(* IEC 61131-3 sources: kst/tests, 86 files *)

(* ---- f.1.st ---- *)
FUNCTION WEIGH : INT
  VAR_INPUT
    weigh_command : BOOL;
    gross_weight : INT ;
    tare_weight : INT ;
  END_VAR

IF weigh_command THEN
  WEIGH := gross_weight - tare_weight;
END_IF ;
END_FUNCTION

(* ---- f.11.st ---- *)
FUNCTION ALRMINT : BOOL
VAR_INPUT
  IN:INT;
  THI:INT ;
  TLO:INT  ;
END_VAR
VAR_OUTPUT
  HI: BOOL;
  LO: BOOL;
END_VAR
HI := IN > THI ;

LO := IN < THL ;
ALRMINT := THI OR THL ;
END_FUNCTION

(* ---- f10.st ---- *)
FUNCTION SIMPLE_FUN : REAL
    VAR_INPUT
  		A, B : REAL ;
      	C : REAL := 1.0;
  	END_VAR
  	VAR_IN_OUT COUNT : INT ; END_VAR
  	VAR COUNTP1 : INT ; END_VAR

  	COUNTP1 := ADD(COUNT,1);
  	COUNT := COUNTP1 ;
    SIMPLE_FUN := A*B/C;
END_FUNCTION

(* ---- f22.st ---- *)
FUNCTION Test : BOOL
	VAR_INPUT
		SUM : INT;
		FLAG : BOOL;
	END_VAR
	VAR
		I, J : INT;
	END_VAR

	SUM := 0 ;
	FOR I := 1 TO 3 DO
		FOR J := 1 TO 2 DO
			IF FLAG THEN EXIT ; END_IF
			SUM := SUM + J ;
		END_FOR ;
		SUM := SUM + I ;
	END_FOR ;
END_FUNCTION

(* ---- f5.st ---- *)
FUNCTION Test : INT
	VAR_INPUT
		B, C, D : INT;
		X : INT;
	END_VAR
	VAR_OUTPUT
		A : INT;
		NO_ERR : BOOL;
	END_VAR

	A := ADD(B, C, D);
	A := SHL(IN:=B, N:=C);
	A := SHL(EN:=ENABLE, IN:=B, N:=C, NOT ENO=>NO_ERR);
	A := INC(V:=X);

END_FUNCTION

(* ---- t19-1.st ---- *)
FUNCTION Test : INT
	VAR_INPUT
		B, COND, TEMPL : INT;
	END_VAR
	VAR_OUTPUT
		A : INT;
	END_VAR

	A := LIMIT(EN:=COND, IN:=B, MX:=5, ENO=>TEMPL);

END_FUNCTION

(* ---- t19-2.st ---- *)
FUNCTION Test : INT
	VAR_INPUT
		B : INT;
	END_VAR
	VAR_OUTPUT
		A : INT;
	END_VAR

	A := LIMIT(1, B, 5);

END_FUNCTION

(* ---- t20-3a.st ---- *)
FUNCTION SIMPLE_FUN : REAL
    VAR_INPUT
  		A, B : REAL ;
      	C : REAL := 1.0;
  	END_VAR
  	VAR_IN_OUT COUNT : INT ; END_VAR
  	VAR COUNTP1 : INT ; END_VAR

  	COUNTP1 := ADD(COUNT,1);
  	COUNT := COUNTP1 ;
    SIMPLE_FUN := A*B/C;
END_FUNCTION

(* ---- t56-1.st ---- *)
FUNCTION Test : INT
	VAR_INPUT
		B : INT;
	END_VAR
	VAR_OUTPUT
		A, CV : INT;
		C : REAL;
	END_OUTPUT

	A := B;
	CV := CV+1;
	C := SIN(X);

END_FUNCTION

(* ---- t56-4.st ---- *)
FUNCTION Test : BOOL
	VAR_INPUT
		A, B, C : REAL;
	END_VAR
	VAR_OUTPUT
		D, X1, X2 : REAL;
		NROOTS : INT;
	END_VAR

	D := B*B - 4*A*C ;
	IF D < 0.0 THEN NROOTS := 0 ;
	ELSIF D = 0.0 THEN
		NROOTS := 1 ;
		X1 := - B/(2.0*A) ;
	ELSE
		NROOTS := 2 ;
		X1 := (- B + SQRT(D))/(2.0*A) ;
		X2 := (- B - SQRT(D))/(2.0*A) ;
	END_IF ;
END_FUNCTION

(* ---- t56-6.st ---- *)
FUNCTION Test : BOOL
	VAR_INPUT
		I, J : INT;
	END_VAR

	J := 101 ;
	FOR I := 1 TO 100 BY 2 DO
		IF I MOD 2 == 0 THEN
			J := I ;
			EXIT ;
		END_IF ;
	END_FOR ;
END_FUNCTION

(* ---- t56-7.st ---- *)
FUNCTION Test : BOOL
	VAR_INPUT
		J : INT;
	END_VAR

	J := 1;
	WHILE J <= 100 DO
		J := J+2 ;
	END_WHILE ;
END_FUNCTION

(* ---- t56-8.st ---- *)
FUNCTION Test : BOOL
	VAR_INPUT
		J : INT;
	END_VAR

	J := -1 ;
	REPEAT
	  J := J+2 ;
	UNTIL J = 101
	END_REPEAT ;
END_FUNCTION

(* ---- f.2.st ---- *)
FUNCTION_BLOCK CMD_MONITOR
 VAR_INPUT AUTO_CMD : BOOL ;
          AUTO_MODE : BOOL ;
            MAN_CMD : BOOL ;
        MAN_CMD_CHK : BOOL ;
          T_CMD_MAX : REAL ;
               FDBK : BOOL ;
                ACK : BOOL ;
 END_VAR
 VAR_OUTPUT CMD : BOOL ;
           ALRM : BOOL ;
 END_VAR
 VAR CMD_TMR : TON ;
     ALRM_FF : SR ;
 END_VAR

 CMD := AUTO_CMD & AUTO_MODE
          OR MAN_CMD & NOT MAN_CMD_CHK & NOT AUTO_MODE ;
    CMD_TMR (IN := CMD, PT := T_CMD_MAX);
    ALRM_FF (S1 := CMD_TMR.Q & NOT FDBK, R := ACK);
    ALRM := ALRM_FF.Q1;

END_FUNCTION_BLOCK

(* ---- f.3.st ---- *)
FUNCTION_BLOCK FWD_REV_MON
VAR_INPUT AUTO : BOOL ;
  ACK : BOOL ;
  AUTO_FWD : BOOL ;
  MAN_FWD : BOOL ;
  MAN_FWD_CHK : BOOL ;
  T_FWD_MAX : TIME ;
  FWD_FDBK : BOOL ;

  AUTO_REV : BOOL ;
  MAN_REV : BOOL ;
  MAN_REV_CHK : BOOL ;
  T_REV_MAX : TIME ;
  REV_FDBK : BOOL ;
END_VAR
VAR_OUTPUT KLAXON : BOOL ;
  FWD_REV_ALRM : BOOL;
  FWD_CMD : BOOL ;
  FWD_ALRM : BOOL ;
  REV_CMD : BOOL ;
  REV_ALRM : BOOL ;
END_VAR
VAR FWD_MON : CMD_MONITOR;
  REV_MON : CMD_MONITOR;
  FWD_REV_FF : SR ;
END_VAR

  FWD_MON    (AUTO_MODE   := AUTO,
              ACK         := ACK,
              AUTO_CMD    := AUTO_FWD,
              MAN_CMD     := MAN_FWD,
              MAN_CMD_CHK := MAN_FWD_CHK,
              T_CMD_MAX   := T_FWD_MAX,
              FDBK        := FWD_FDBK);
  REV_MON    (AUTO_MODE   := AUTO,
              ACK         := ACK,
              AUTO_CMD    := AUTO_REV,
              MAN_CMD     := MAN_REV,
              MAN_CMD_CHK := MAN_REV_CHK,
              T_CMD_MAX   := T_REV_MAX,
              FDBK        := REV_FDBK);
  FWD_REV_FF (S1 := FWD_MON.CMD & REV_MON.CMD, R := ACK);

  FWD_REV_ALRM := FWD_REV_FF.Q1;
  FWD_CMD := FWD_MON.CMD & NOT FWD_REV_ALRM;
  FWD_ALRM := FWD_MON.ALRM;
  REV_CMD := REV_MON.CMD & NOT FWD_REV_ALRM;
  REV_ALRM := REV_MON.ALRM;
  KLAXON := FWD_ALRM OR REV_ALRM OR FWD_REV_ALRM;
END_FUNCTION_BLOCK

(* ---- f.4.st ---- *)
FUNCTION_BLOCK STACK_INT
  VAR_INPUT PUSH, POP: BOOL;
            R1 : BOOL ;
            IN : INT ;
            N  : INT ;
  END_VAR
  VAR_OUTPUT EMPTY : BOOL := 1 ;
             OFLO  : BOOL := 0 ;
             OUT   : INT  := 0 ;
  END_VAR
  VAR STK : ARRAY[0..127] OF INT;
      NI : INT :=128  ;
      PTR : INT := -1 ;
  END_VAR

    IF R1 THEN
       OFLO := 0; EMPTY := 1; PTR := -1;
       NI := LIMIT (MN:=1,IN:=N,MX:=128); OUT := 0;
    ELSIF POP & NOT EMPTY THEN
       OFLO := 0; PTR := PTR-1; EMPTY := PTR < 0;
       IF EMPTY THEN OUT := 0;
       ELSE OUT := STK[PTR];
       END_IF ;
    ELSIF PUSH & NOT OFLO THEN
       EMPTY := 0; PTR := PTR+1; OFLO := (PTR = NI);
       IF NOT OFLO THEN OUT := IN ; STK[PTR] := IN;
       ELSE OUT := 0;
       END_IF ;
    END_IF ;
END_FUNCTION_BLOCK

(* ---- f.6.1.st ---- *)
FUNCTION_BLOCK LAG1
   VAR_INPUT
     RUN : BOOL ;
     XIN : REAL ;
     TAU : REAL ;
     CYCLE : REAL ;
   END_VAR
   VAR_OUTPUT XOUT : REAL ; END_VAR
   VAR K : REAL ;
   END_VAR
   IF RUN THEN XOUT := XOUT + K * (XIN - XOUT) ;
   ELSE XOUT := XIN ;
        K := CYCLE /(CYCLE + TAU) ;
   END_IF ;
END_FUNCTION_BLOCK

(* ---- f.6.10.st ---- *)
FUNCTION_BLOCK PID
   VAR_INPUT
     AUTO : BOOL ;
     PV : REAL ;
     SP : REAL ;
     X0 : REAL ;

     KP : REAL ;
     TR : REAL ;
     TD : REAL ;
     CYCLE : REAL ;
   END_VAR
   VAR_OUTPUT XOUT : REAL; END_VAR
   VAR ERROR : REAL ;
       ITERM : INTEGRAL ;
       DTERM : DERIVATIVE ;
   END_VAR
   ERROR := PV - SP ;

   ITERM (RUN := AUTO, R1 := NOT AUTO, XIN := ERROR,
          X0 := TR * (X0 - ERROR), CYCLE := CYCLE) ;
   DTERM (RUN := AUTO, XIN := ERROR, CYCLE := CYCLE) ;
   XOUT := KP * (ERROR + ITERM.XOUT/TR + DTERM.XOUT*TD) ;
 END_FUNCTION_BLOCK

(* ---- f.6.11.st ---- *)
FUNCTION_BLOCK DIFFEQ
   VAR_INPUT
     RUN : BOOL ;
     XIN : REAL ;
     A : ARRAY[1..127] OF REAL ;
     M : INT ;
     B : ARRAY[0..127] OF REAL ;
     N : INT ;
   END_VAR
   VAR_OUTPUT XOUT : REAL := 0.0 ; END_VAR
   VAR
     XI : ARRAY [0..127] OF REAL ;
     XO : ARRAY [0..127] OF REAL ;
     I : INT ;
   END_VAR
   XO[0] := XOUT ; XI[0] := XIN ;
   XOUT := B[0] * XIN ;
   IF RUN THEN
      FOR I := M TO 1 BY -1 DO
          XOUT := XOUT + A[I] * XO[I] ; XO[I] := XO[I-1];
      END_FOR;
      FOR I := N TO 1 BY -1 DO
          XOUT := XOUT + B[I] * XI[I] ; XI[I] := XI[I-1];
      END_FOR;
   ELSE
      FOR I := 1 TO M DO XO[I] := 0.0; END_FOR;
      FOR I := 1 TO N DO XI[I] := 0.0; END_FOR;
   END_IF ;
 END_FUNCTION_BLOCK

(* ---- f.6.12.st ---- *)
 FUNCTION_BLOCK RAMP
   VAR_INPUT
     RUN : BOOL ;
     X0,X1 : REAL ;
     TR : REAL ;
     CYCLE : REAL ;
   END_VAR
   VAR_OUTPUT
     BUSY : BOOL ;
     XOUT : REAL := 0.0 ;
   END_VAR
   VAR XI : REAL ;
       T : REAL := 0.0;
   END_VAR
   BUSY := RUN ;
   IF RUN THEN
      IF T >= TR THEN BUSY := 0 ; XOUT := X1 ;
      ELSE XOUT := XI + (X1-XI) * T
                                / TR ;
           T := T + CYCLE ;
      END_IF ;
   ELSE XOUT := X0 ; XI := X0 ; T := 0.0 ;
   END_IF ;
 END_FUNCTION_BLOCK

(* ---- f.6.13.st ---- *)
FUNCTION_BLOCK TRANSFER
 VAR_INPUT
   AUTO : BOOL ;
   XIN : REAL ;
   FASTRATE, SLOWRATE : REAL ;
   FASTUP, SLOWUP,
   FASTDOWN, SLOWDOWN : BOOL;
   CYCLE : TIME ;
 END_VAR
 VAR_OUTPUT XOUT : REAL ; END_VAR
 VAR XFERRAMP : INTEGRAL ;
     RAMPRATE : REAL ;
 END_VAR
 RAMPRATE := 0.0 ;
 IF NOT AUTO THEN
  IF FASTUP THEN RAMPRATE := FASTRATE; END_IF;
  IF SLOWUP THEN RAMPRATE := RAMPRATE + SLOWRATE; END_IF;
  IF FASTDOWN THEN RAMPRATE := RAMPRATE - FASTRATE; END_IF;
  IF SLOWDOWN THEN RAMPRATE := RAMPRATE - SLOWRATE; END_IF;
 END_IF ;
 XFERRAMP (RUN := 1, CYCLE := CYCLE, R1 := AUTO,
            XIN := RAMPRATE, X0 := XIN) ;
 XOUT := XFERRAMP.XOUT;
END_FUNCTION_BLOCK

(* ---- f.6.2.st ---- *)
FUNCTION_BLOCK DELAY
  VAR_INPUT
    RUN : BOOL ;
    XIN : REAL ;
    N   : INT ;
  END_VAR
  VAR_OUTPUT XOUT : REAL; END_VAR
  VAR X : ARRAY [0..127]
               OF REAL;
      I, IXIN, IXOUT : INT := 0;
  END_VAR
  IF RUN THEN IXIN := MOD(IXIN + 1, 128) ; X[IXIN] := XIN ;
              IXOUT := MOD(IXOUT + 1, 128) ; XOUT := X[IXOUT];
  ELSE XOUT := XIN ; IXIN := N ; IXOUT := 0;
       FOR I := 0 TO N DO X[I] := XIN; END_FOR;
  END_IF ;
END_FUNCTION_BLOCK

(* ---- f.6.3.st ---- *)
FUNCTION_BLOCK AVERAGE
   VAR_INPUT
     RUN : BOOL ;
     XIN : REAL ;
     N   : INT ;
   END_VAR
   VAR_OUTPUT XOUT : REAL ; END_VAR
   VAR SUM  : REAL := 0.0;
       FIFO : DELAY ;
   END_VAR
   SUM := SUM - FIFO.XOUT ;
   FIFO (RUN := RUN , XIN := XIN, N := N) ;
   SUM := SUM + FIFO.XOUT ;
   IF RUN THEN XOUT := SUM/N ;
   ELSE SUM := N*XIN ; XOUT := XIN ;
   END_IF ;
 END_FUNCTION_BLOCK

(* ---- f.6.4.st ---- *)
FUNCTION_BLOCK INTEGRAL
   VAR_INPUT
     RUN : BOOL ;
     R1 : BOOL ;
     XIN : REAL ;
     X0  : REAL ;
     CYCLE : REAL ;
   END_VAR
   VAR_OUTPUT
     Q : BOOL ;
     XOUT : REAL ;
   END_VAR
   Q := NOT R1 ;
   IF R1 THEN XOUT := X0 ;
   ELSIF RUN THEN XOUT := XOUT + XIN * TIME_TO_REAL(CYCLE);
   END_IF ;
 END_FUNCTION_BLOCK

(* ---- f.6.5.st ---- *)
FUNCTION_BLOCK DERIVATIVE
   VAR_INPUT
     RUN : BOOL ;
     XIN : REAL ;
     CYCLE : REAL ;
   END_VAR
   VAR_OUTPUT
     XOUT : REAL ;
   END_VAR
   VAR X1, X2, X3 : REAL ; END_VAR
   IF RUN THEN
      XOUT := (3.0 * (XIN - X3) + X1 - X2)
              / (10.0 * CYCLE) ;
      X3 := X2 ; X2 := X1 ; X1 := XIN ;
   ELSE XOUT := 0.0; X1 := XIN ; X2 := XIN ; X3 := XIN ;
   END_IF ;
 END_FUNCTION_BLOCK

(* ---- f.6.6.st ---- *)
 FUNCTION_BLOCK HYSTERESIS
  VAR_INPUT XIN1, XIN2, EPS : REAL; END_VAR
  VAR_OUTPUT Q : BOOL := 0; END_VAR
  IF Q THEN IF XIN1 < (XIN2 - EPS) THEN Q := 0; END_IF ;
  ELSIF XIN1 > (XIN2 + EPS) THEN Q := 1 ;
  END_IF ;
END_FUNCTION_BLOCK

(* ---- f19.st ---- *)
FUNCTION_BLOCK A
	VAR_OUTPUT
		y1 : UINT ; y2 : BYTE ;
	END_VAR
END_FUNCTION_BLOCK

FUNCTION_BLOCK B
	VAR_INPUT
		b1 : UINT ; b2 : BYTE ;
	END_VAR
END_FUNCTION_BLOCK

FUNCTION_BLOCK C
	VAR_OUTPUT c1 : BOOL ; END_VAR
	VAR C2 AT %Q*: BYTE;
		C3: INT;
	END_VAR
END_FUNCTION_BLOCK

FUNCTION_BLOCK D
	VAR_INPUT d1 : BOOL ; END_VAR
	VAR_OUTPUT y2 : INT ; END_VAR
END_FUNCTION_BLOCK

PROGRAM F
	VAR_INPUT  x1 : BOOL ;  x2 : UINT ; END_VAR
	VAR_OUTPUT y1 : BYTE ; END_VAR
	VAR COUNT: INT; TIME1: TON; END_VAR
END_PROGRAM

PROGRAM G
	VAR_OUTPUT out1 : UINT ;  END_VAR
	VAR_EXTERNAL z1 : BYTE ;  END_VAR
	VAR  FB1 : A ;  FB2 : B ; END_VAR
	FB1();
	out1 := FB1.y1;
	z1 := FB1.y2;
    FB2(b1 := FB1.y1, b2 := FB1.y2) ;
END_PROGRAM

PROGRAM H
	VAR_OUTPUT HOUT1: INT ;  END_VAR
	VAR  FB1 : C ;  FB2 : D ; END_VAR
	FB1();
	FB2(d1:=TRUE);
	HOUT1 := FB2.y2;
END_PROGRAM

(* ---- hc-t-171.st ---- *)
PROGRAM temp
  VAR
    I1,I2,I3,I4:INT;
    B1,B2,B3,B4,B5,B6,B7:BOOL;
    R1,R2,R3,R4:REAL;
  END_VAR

  CMD_MONITOR(AUTO_CMD:=B1,AUTO_MODE:=B2,MAN_CMD:=B3,MAN_CMD_CHK:=B4,FDBK:=B5,ACK:=B6,T_CMD_MAX:=R1);

END_PROGRAM

FUNCTION_BLOCK CMD_MONITOR
 VAR_INPUT AUTO_CMD : BOOL ;
          AUTO_MODE : BOOL ;
            MAN_CMD : BOOL ;
        MAN_CMD_CHK : BOOL ;
          T_CMD_MAX : REAL ;
               FDBK : BOOL ;
                ACK : BOOL ;
 END_VAR
 VAR_OUTPUT CMD : BOOL ;
           ALRM : BOOL ;
 END_VAR
 VAR CMD_TMR : TON ;
     ALRM_FF : SR ;
 END_VAR

 CMD := AUTO_CMD & AUTO_MODE
          OR MAN_CMD & NOT MAN_CMD_CHK & NOT AUTO_MODE ;
    CMD_TMR (IN := CMD, PT := T_CMD_MAX);
    ALRM_FF (S1 := CMD_TMR.Q & NOT FDBK, R := ACK);
    ALRM := ALRM_FF.Q1;

END_FUNCTION_BLOCK

(* ---- hc-t-178.st ---- *)
PROGRAM temp
  VAR
    I1,I2,I3,I4:INT;
    B1,B2,B3:BOOL;
    R0,R2,R3,R4:REAL;
  END_VAR

  STACK_INT(PUSH:=B1,POP:=B2,R1:=B3,IN:=I1,N:=I2);

END_PROGRAM

FUNCTION_BLOCK STACK_INT
  VAR_INPUT PUSH, POP: BOOL R_EDGE;
            R1 : BOOL ;
            IN : INT ;
            N  : INT ;
  END_VAR
  VAR_OUTPUT EMPTY : BOOL := 1 ;
             OFLO  : BOOL := 0 ;
             OUT   : INT  := 0 ;
  END_VAR
  VAR STK : ARRAY[0..127] OF INT;
      NI : INT :=128  ;
      PTR : INT := -1 ;
  END_VAR

    IF R1 THEN
       OFLO := 0; EMPTY := 1; PTR := -1;
       NI := LIMIT (MN:=1,IN:=N,MX:=128); OUT := 0;
    ELSIF POP & NOT EMPTY THEN
       OFLO := 0; PTR := PTR-1; EMPTY := PTR < 0;
       IF EMPTY THEN OUT := 0;
       ELSE OUT := STK[PTR];
       END_IF ;
    ELSIF PUSH & NOT OFLO THEN
       EMPTY := 0; PTR := PTR+1; OFLO := (PTR = NI);
       IF NOT OFLO THEN OUT := IN ; STK[PTR] := IN;
       ELSE OUT := 0;
       END_IF ;
    END_IF ;
END_FUNCTION_BLOCK

(* ---- hc-t-187.st ---- *)
PROGRAM temp
  VAR
    I1,I2,I3,I4:INT;
    B1,B2,B3:BOOL;
    R1,R2,R3,R4:REAL;
  END_VAR

  LAG1(RUN:=B1,XIN:=R1,TAU:=R2,CYCLE:=R3)
  DELAY(RUN:=B1,XIN:=R1,TAU:=R2,CYCLE:=R3)

END_PROGRAM

FUNCTION_BLOCK LAG1
   VAR_INPUT
     RUN : BOOL ;
     XIN : REAL ;
     TAU : REAL ;
     CYCLE : REAL ;
   END_VAR
   VAR_OUTPUT XOUT : REAL ; END_VAR
   VAR K : REAL ;
   END_VAR
   IF RUN THEN XOUT := XOUT + K * (XIN - XOUT) ;
   ELSE XOUT := XIN ;
        K := CYCLE /(CYCLE + TAU) ;
   END_IF ;
 END_FUNCTION_BLOCK

 FUNCTION_BLOCK DELAY
  VAR_INPUT
    RUN : BOOL ;
    XIN : REAL ;
    N   : INT ;
  END_VAR
  VAR_OUTPUT XOUT : REAL; END_VAR
  VAR X : ARRAY [0..127]
               OF REAL;
      I, IXIN, IXOUT : INT := 0;
  END_VAR
  IF RUN THEN IXIN := MOD(IXIN + 1, 128) ; X[IXIN] := XIN ;
              IXOUT := MOD(IXOUT + 1, 128) ; XOUT := X[IXOUT];
  ELSE XOUT := XIN ; IXIN := N ; IXOUT := 0;
       FOR I := 0 TO N DO X[I] := XIN; END_FOR;
  END_IF ;
END_FUNCTION_BLOCK

(* ---- hc-t-188.st ---- *)
PROGRAM temp
  VAR
    I1,I2,I3,I4:INT;
    B1,B2,B3:BOOL;
    R0,R2,R3,R4:REAL;
  END_VAR

  AVERAGE(RUN:=B1,XIN:=R0,N:=I1);
  INTEGRAL(RUN:=B1,R1:=B2,XIN:=R0,X0:=R2,CYCLE:=R43);

END_PROGRAM

FUNCTION_BLOCK AVERAGE
   VAR_INPUT
     RUN : BOOL ;
     XIN : REAL ;
     N   : INT ;
   END_VAR
   VAR_OUTPUT XOUT : REAL ; END_VAR
   VAR SUM  : REAL := 0.0;
       FIFO : DELAY ;
   END_VAR
   SUM := SUM - FIFO.XOUT ;
   FIFO (RUN := RUN , XIN := XIN, N := N) ;
   SUM := SUM + FIFO.XOUT ;
   IF RUN THEN XOUT := SUM/N ;
   ELSE SUM := N*XIN ; XOUT := XIN ;
   END_IF ;
 END_FUNCTION_BLOCK

FUNCTION_BLOCK INTEGRAL
   VAR_INPUT
     RUN : BOOL ;
     R1 : BOOL ;
     XIN : REAL ;
     X0  : REAL ;
     CYCLE : REAL ;
   END_VAR
   VAR_OUTPUT
     Q : BOOL ;
     XOUT : REAL ;
   END_VAR
   Q := NOT R1 ;
   IF R1 THEN XOUT := X0 ;
   ELSIF RUN THEN XOUT := XOUT + XIN * TIME_TO_REAL(CYCLE);
   END_IF ;
 END_FUNCTION_BLOCK

(* ---- hc-t-189.st ---- *)
PROGRAM temp
  VAR
    I1,I2,I3,I4:INT;
    B1,B2,B3:BOOL;
    R1,R2,R3,R4:REAL;
  END_VAR
  DERIVATIVE(RUN:=B1,XIN:=R1,CYCLE:=R2);
  HYSTERESIS(XIN1:=R3,XIN2:=R4,EPS:=R5);
END_PROGRAM

FUNCTION_BLOCK DERIVATIVE
   VAR_INPUT
     RUN : BOOL ;
     XIN : REAL ;
     CYCLE : REAL ;
   END_VAR
   VAR_OUTPUT
     XOUT : REAL ;
   END_VAR
   VAR X1, X2, X3 : REAL ; END_VAR
   IF RUN THEN
      XOUT := (3.0 * (XIN - X3) + X1 - X2)
              / (10.0 * CYCLE) ;
      X3 := X2 ; X2 := X1 ; X1 := XIN ;
   ELSE XOUT := 0.0; X1 := XIN ; X2 := XIN ; X3 := XIN ;
   END_IF ;
 END_FUNCTION_BLOCK

 FUNCTION_BLOCK HYSTERESIS
  VAR_INPUT XIN1, XIN2, EPS : REAL; END_VAR
  VAR_OUTPUT Q : BOOL := 0; END_VAR
  IF Q THEN IF XIN1 < (XIN2 - EPS) THEN Q := 0; END_IF ;
  ELSIF XIN1 > (XIN2 + EPS) THEN Q := 1 ;
  END_IF ;
END_FUNCTION_BLOCK

(* ---- hc-t-192.st ---- *)
PROGRAM temp
  VAR
    I1,I2,I3,I4:INT;
    B1,B2,B3:BOOL;
    R1,R2,R3,R4,R5,R6,R7:REAL;
  END_VAR

  PID(AUTO:=B1,PV:=R1,SP:=R2,X0:=R3,KP:=R4,TR:=R5,TD:=R6,CYCLE:=R7);

END_PROGRAM

FUNCTION_BLOCK PID
   VAR_INPUT
     AUTO : BOOL ;
     PV : REAL ;
     SP : REAL ;
     X0 : REAL ;

     KP : REAL ;
     TR : REAL ;
     TD : REAL ;
     CYCLE : REAL ;
   END_VAR
   VAR_OUTPUT XOUT : REAL; END_VAR
   VAR ERROR : REAL ;
       ITERM : INTEGRAL ;
       DTERM : DERIVATIVE ;
   END_VAR
   ERROR := PV - SP ;

   ITERM (RUN := AUTO, R1 := NOT AUTO, XIN := ERROR,
          X0 := TR * (X0 - ERROR), CYCLE := CYCLE) ;
   DTERM (RUN := AUTO, XIN := ERROR, CYCLE := CYCLE) ;
   XOUT := KP * (ERROR + ITERM.XOUT/TR + DTERM.XOUT*TD) ;
 END_FUNCTION_BLOCK

(* ---- hc-t-193.st ---- *)
PROGRAM temp
  VAR
    P1,P2:INT;
    P3:REAL;
    P4:BOOL;
  END_VAR

  DIFFEQ(RUN:=P4,XIN:=P3);

END_PROGRAM

FUNCTION_BLOCK DIFFEQ
   VAR_INPUT
     RUN : BOOL ;
     XIN : REAL ;
     A : ARRAY[1..127] OF REAL ;
     M : INT ;
     B : ARRAY[0..127] OF REAL ;
     N : INT ;
   END_VAR
   VAR_OUTPUT XOUT : REAL := 0.0 ; END_VAR
   VAR
     XI : ARRAY [0..127] OF REAL ;
     XO : ARRAY [0..127] OF REAL ;
     I : INT ;
   END_VAR
   XO[0] := XOUT ; XI[0] := XIN ;
   XOUT := B[0] * XIN ;
   IF RUN THEN
      FOR I := M TO 1 BY -1 DO
          XOUT := XOUT + A[I] * XO[I] ; XO[I] := XO[I-1];
      END_FOR;
      FOR I := N TO 1 BY -1 DO
          XOUT := XOUT + B[I] * XI[I] ; XI[I] := XI[I-1];
      END_FOR;
   ELSE
      FOR I := 1 TO M DO XO[I] := 0.0; END_FOR;
      FOR I := 1 TO N DO XI[I] := 0.0; END_FOR;
   END_IF ;
 END_FUNCTION_BLOCK

(* ---- hc-t-194.st ---- *)
PROGRAM temp
  VAR
    I1,I2,I3,I4:INT;
    B1,B2,B3:BOOL;
    R1,R2,R3,R4:REAL;
  END_VAR
  RAMP(RUN:=B1,X0:=R1,X1:=R2,TR:=R3,CYCLE:=R4);

END_PROGRAM

 FUNCTION_BLOCK RAMP
   VAR_INPUT
     RUN : BOOL ;
     X0,X1 : REAL ;
     TR : REAL ;
     CYCLE : REAL ;
   END_VAR
   VAR_OUTPUT
     BUSY : BOOL ;
     XOUT : REAL := 0.0 ;
   END_VAR
   VAR XI : REAL ;
       T : REAL := 0.0;
   END_VAR
   BUSY := RUN ;
   IF RUN THEN
      IF T >= TR THEN BUSY := 0 ; XOUT := X1 ;
      ELSE XOUT := XI + (X1-XI) * T
                                / TR ;
           T := T + CYCLE ;
      END_IF ;
   ELSE XOUT := X0 ; XI := X0 ; T := 0.0 ;
   END_IF ;
 END_FUNCTION_BLOCK

(* ---- SR.st ---- *)
FUNCTION_BLOCK SR
	VAR_INPUT
		S1, R : BOOL;
	END_VAR
	VAR_OUTPUT
		Q1 : BOOL;
	END_VAR

	Q1 := S1 XOR (Q1 AND NOT R);
END_FUNCTION_BLOCK

(* ---- t33-11.st ---- *)
FUNCTION_BLOCK AND_EDGE
	VAR INPUT X : BOOL; Y : BOOL; END_VAR
    VAR X_TRIG : R_TRIG ; Y_TRIG : F_TRIG ; END_VAR

    X_TRIG(CLK := X) ;
	Y_TRIG(CLK := Y) ;
    Z := X_TRIG.Q AND Y_TRIG.Q;
END_FUNCTION_BLOCK

(* ---- t33-12a.st ---- *)
FUNCTION_BLOCK ACCUM
   VAR_IN_OUT A : INT ; END_VAR
   VAR_INPUT X : INT ; END_VAR
   A := A+X ;
END_FUNCTION_BLOCK

(* ---- t33-12b.st ---- *)
FUNCTION_BLOCK ACCUM
   VAR
	    ACC : INT ;
	    X1  : INT ;
	    X2  : INT ;
	END_VAR
	ACC := ACC+X1*X2 ;
END_FUNCTION_BLOCK

(* ---- t33-12c.st ---- *)
FUNCTION_BLOCK ACCUM
   VAR
	    ACC : INT ;
	    X1  : INT ;
	    X2  : INT ;
	    X3  : INT ;
	END_VAR
	ACC := ACC+X1*X2+X3*X4;
END_FUNCTION_BLOCK

(* ---- t33-12d.st ---- *)
FUNCTION_BLOCK ACCUM
   VAR
		X1  : INT ;
	    X2  : INT ;
	    X3  : INT ;
	    X4  : INT ;
	END_VAR

	X3 := X3+X1*X2 ;
	X4 := X3 ;
END_FUNCTION_BLOCK

(* ---- t33-1a.st ---- *)
FUNCTION_BLOCK Test
	VAR RETAIN X : REAL ; END_VAR
END_FUNCTION_BLOCK

(* ---- t33-1b.st ---- *)
FUNCTION_BLOCK Test
	VAR NON_RETAIN X : REAL ; END_VAR
END_FUNCTION_BLOCK

(* ---- t33-2a.st ---- *)
FUNCTION_BLOCK Test
	VAR_OUTPUT RETAIN X : REAL ; END_VAR
END_FUNCTION_BLOCK

(* ---- t33-2b.st ---- *)
FUNCTION_BLOCK Test
	VAR_INPUT RETAIN X : REAL ; END_VAR
END_FUNCTION_BLOCK

(* ---- t33-2c.st ---- *)
FUNCTION_BLOCK Test
	VAR_OUTPUT NON_RETAIN X : REAL ; END_VAR
END_FUNCTION_BLOCK

(* ---- t33-2d.st ---- *)
FUNCTION_BLOCK Test
	VAR_INPUT NON_RETAIN X : REAL ; END_VAR
END_FUNCTION_BLOCK

(* ---- t33-3a.st ---- *)
FUNCTION_BLOCK Test
	VAR RETAIN TMR1: TON ; END_VAR
END_FUNCTION_BLOCK

(* ---- t33-3b.st ---- *)
FUNCTION_BLOCK Test
	VAR NON_RETAIN TMR1: TON ; END_VAR
END_FUNCTION_BLOCK

(* ---- t33-4a.st ---- *)
FUNCTION_BLOCK Test
	VAR_IN_OUT A: INT ; END_VAR
END_FUNCTION_BLOCK

(* ---- t33-5a.st ---- *)
FUNCTION_BLOCK Test
	VAR
		EXPIRED : BOOL;
	END_VAR
	VAR_INPUT I_TMR: TON ; END_VAR

	EXPIRED := I_TMR.Q;
END_FUNCTION_BLOCK

(* ---- t33-6a.st ---- *)
FUNCTION_BLOCK Test
	VAR EXPIRED : BOOL END_VAR
	VAR_IN_OUT IO_TMR: TOF ; END_VAR

	IO_TMR(IN:=A_VAR, PT:=T#10S);
	EXPIRED := IO_TMR.Q;
END_FUNCTION_BLOCK

(* ---- t33-7a.st ---- *)
FUNCTION_BLOCK Test
	VAR EXPIRED : BOOL END_VAR
	VAR_EXTERNAL EX_TMR : TOF ;END_VAR

	EX_TMR(IN:=A_VAR,  PT:=T#10S);
	EXPIRED := EX_TMR.Q;
END_FUNCTION_BLOCK

(* ---- t33-8a.st ---- *)
FUNCTION_BLOCK AND_EDGE
	VAR_INPUT X : BOOL R_EDGE;
	          Y : BOOL F_EDGE;
	END_VAR
	VAR_OUTPUT Z : BOOL ; END_VAR
	Z := X AND Y ;
END_FUNCTION_BLOCK

(* ---- t35-1.st ---- *)
FUNCTION_BLOCK R_TRIG
    VAR_INPUT  CLK: BOOL; END_VAR
    VAR_OUTPUT  Q: BOOL; END_VAR
    VAR M: BOOL; END_VAR

	Q := CLK AND NOT M;
	M := CLK;
END_FUNCTION_BLOCK

(* ---- t35-2.st ---- *)
FUNCTION_BLOCK F_TRIG
    VAR_INPUT  CLK: BOOL; END_VAR
    VAR_OUTPUT   Q: BOOL; END_VAR
    VAR M: BOOL; END_VAR

	Q := NOT CLK AND NOT M;
	M := NOT CLK;
END_FUNCTION_BLOCK

(* ---- t36-1a.st ---- *)
FUNCTION_BLOCK F_TRIG
	VAR_INPUT
		R, CU : BOOL;
		PV : INT;
	END_VAR
	VAR_OUT
		CV : INT;
		Q : BOOL;
	END_VAR;
	VAR
		PVmax : INT;
	END_VAR

	IF R THEN CV := 0 ;
	ELSIF CU AND (CV < PVmax)
	    THEN CV := CV+1;
	END_IF ;
	Q := (CV >= PV) ;

END_FUNCTION_BLOCK

(* ---- t36-2a.st ---- *)
FUNCTION_BLOCK F_TRIG
	VAR_INPUT
		LD, CD : BOOL;
		PV : INT;
	END_VAR
	VAR_OUT
		CV : INT;
		Q : BOOL;
	END_VAR;
	VAR
		PVmin : INT;
	END_VAR

	IF LD THEN CV := PV ;
	ELSIF CD AND (CV > PVmin)
	THEN CV := CV-1;
	END_IF ;
	Q := (CV <= 0) ;

END_FUNCTION_BLOCK

(* ---- t36-3a.st ---- *)
FUNCTION_BLOCK F_TRIG
	VAR_INPUT
		CU, CD, R, LD: BOOL;
		PV : INT;
	END_VAR
	VAR_OUT
		CV : INT;
		QU, QD : BOOL;
	END_VAR;
	VAR
		PVmax, PVmin : INT;
	END_VAR
	IF R THEN CV := 0 ;
	ELSIF LD THEN CV := PV ;
	ELSE
		IF NOT (CU AND CD) THEN
		    IF CU AND (CV < PVmax)
		    THEN CV := CV+1;
		    ELSIF CD AND (CV > PVmin)
		    THEN CV := CV-1;
		    END_IF;
		END_IF;
	END_IF ;
	QU := (CV >= PV) ;
	QD := (CV <= 0) ;
END_FUNCTION_BLOCK

(* ---- t56-2.st ---- *)
FUNCTION_BLOCK FB
	VAR_INPUT
		IN : INT;
		PT : TIME;
	END_VAR
	VAR_OUTPUT
		Q : BOOL;
	END_VAR

END_FUNCTION_BLOCK

FUNCTION_BLOCK Test
	VAR
		CMD_TMR : FB;
		A : BOOl;
	END_VAR

	CMD_TMR(IN:=%IX5, PT:=T#300ms) ;
	A := CMD_TMR.Q ;

END_FUNCTION_BLOCK

(* ---- TON.st ---- *)
FUNCTION_BLOCK TON
	VAR_INPUT
		IN : BOOL;
		PT : TIME;
	END_VAR
	VAR_OUTPUT
		Q : BOOL;
		ET : TIME;
	END_VAR
	VAR
		RUNNING : BOOL;
		START : TIME;
	END_VAR

	IF IN = FALSE THEN
		Q := FALSE;
		ET := 0;
		RUNNING := FALSE;
	ELSIF RUNNING = FALSE THEN
		START := CTIME;
		RUNNING := TRUE;
	ELSIF CTIME - (START + PT) >= 0 THEN
		Q := TRUE;
		ET := PT;
	ELSE
		IF not Q THEN
			ET := CTIME - START;
		END_IF;
	END_IF;
END_FUNCTION_BLOCK

(* ---- bool.st ---- *)
PROGRAM Bool
	VAR
		X : BOOL := TRUE;
	END_VAR

	X := NOT X;
END_PROGRAM

(* ---- counter.st ---- *)
PROGRAM Counter
	VAR
		A : INT;
		Counter : INT := 5;
	END_VAR
	A := 0;
	A := Inc(In:=Counter, Out=>Counter) + Dec(In:=Counter, Out=>Counter);
	@ltlmc : L

END_PROGRAM

FUNCTION Inc : INT
	VAR_INPUT
		In : INT;
	END_VAR
	VAR_OUTPUT
		Out : INT;
	END_VAR

	Out := In + 1;
	Inc := In;

END_FUNCTION

FUNCTION Dec : INT
	VAR_INPUT
		In : INT;
	END_VAR
	VAR_OUTPUT
		Out : INT;
	END_VAR

	Out := In - 1;
	Dec := In;

END_FUNCTION

// krun -d build --ltlmc "[]Ltl (<>Ltl eqTo(Counter:::A, 7))" tests\counter.st
// krun -d build --ltlmc "[]Ltl (<>Ltl eqTo(Counter:::A, 11))" tests\counter.st

(* ---- fibonacci-numbers.st ---- *)
PROGRAM Fibonacci
  VAR_INPUT
    N : INT := 5;
  END_VAR
  VAR_OUTPUT
	O : INT := 1;
  END_VAR
  VAR
    F1, F2, CNT : INT;
  END_VAR

  F1 := 1;
  F2 := 1;
  CNT := 2;

  IF N <= CNT THEN
    O := 1;
  ELSE
    WHILE CNT < N DO
      O := AddTwo(In0:=F1, In1:=F2);
      F1 := F2;
      F2 := O;
      CNT := CNT + 1;
    END_WHILE;
  END_IF;

END_PROGRAM

FUNCTION AddTwo : INT
  VAR_INPUT
    In0, In1 : INT;
  END_VAR

  AddTwo := In0 + In1;
END_FUNCTION

(* ---- hc-fibonacci-numbers.st ---- *)
PROGRAM Fibonacci
  VAR_INPUT
    N : INT := 1;
  END_VAR
  VAR_OUTPUT
	O : INT := 1;
  END_VAR
  VAR
    F1, F2, CNT : INT;
  END_VAR

  F1 := 1;
  F2 := 1;
  CNT := 2;

  IF N <= CNT THEN
    O := 1;
  ELSE
    WHILE CNT < N DO
      O := AddTwo(In0:=F1, In1:=F2);
      F1 := F2;
      F2 := O;
      CNT := CNT + 1;
    END_WHILE;
  END_IF;

END_PROGRAM

FUNCTION AddTwo : INT
  VAR_INPUT
    In0, In1 : INT;
  END_VAR

  AddTwo := In0 + In1;
END_FUNCTION

(* ---- hc-t-169.st ---- *)
PROGRAM temp
  VAR
    I1,I2,I3,I4:INT;
    B1,B2,B3:BOOL;
    R1,R2,R3,R4:REAL;
  END_VAR

  I3:=WEIGH(weigh_command:=B1,gross_weight:=I1,tare_weight:=I2);

END_PROGRAM

FUNCTION WEIGH : INT
  VAR_INPUT
    weigh_command : BOOL;
    gross_weight : INT ;
    tare_weight : INT ;
  END_VAR

IF weigh_command THEN
  WEIGH := gross_weight - tare_weight;
END_IF ;
END_FUNCTION

(* ---- hc-t-207.st ---- *)
PROGRAM test207
  VAR
    P1,P2,P3:INT;
    P4:BOOL;
  END_VAR

  P4:=ALRMINT(IN:=P1,THI:=P2,TLO:=P3);

END_PROGRAM

FUNCTION ALRMINT : BOOL
VAR_INPUT
  IN:INT;
  THI:INT ;
  TLO:INT  ;
END_VAR
VAR_OUTPUT
  HI: BOOL;
  LO: BOOL;
END_VAR
HI := IN > THI ;

LO := IN < THL ;
ALRMINT := THI OR THL ;
END_FUNCTION

(* ---- sumc.st ---- *)
PROGRAM Sumc
	VAR
		n, i, s : INT;
	END_VAR

	n := 100;
	WHILE i < n DO
		i := i + 1;
		s := s + i;
		@ltlmc : L
	END_WHILE;
END_PROGRAM

// krun -d build --ltlmc "[]Ltl ( L ->Ltl eqToSum(Sumc:::s, Sumc:::i))" tests\sumc.st

(* ---- t17-1.st ---- *)
PROGRAM Test
	VAR
	    AT %IW6.2 : WORD;
	    AT %MW6   : INT ;
	END_VAR
END_PROGRAM

(* ---- t17-2.st ---- *)
PROGRAM Test
	VAR RETAIN
  		AT %QW5 : WORD ;
	END_VAR
END_PROGRAM

(* ---- t17-3.st ---- *)
PROGRAM Test
	VAR_GLOBAL
 		LIM_SW_S5 AT %IX27 : BOOL;
 		CONV_START AT %QX25 : BOOL;
 		TEMPERATURE AT %IW28: INT;
 		VAR C2 AT %Q* : BYTE ;
	END_VAR
END_PROGRAM

(* ---- t17-4.st ---- *)
PROGRAM Test
	VAR
		INARY AT %IW6 ;
 		ARRAY [0..9] OF INT;
	END_VAR
END_PROGRAM

(* ---- t17-5.st ---- *)
PROGRAM Test
	VAR
		CONDITION_RED : BOOL;
		IBOUNCE : WORD ;
		MYDUB : DWORD ;
		AWORD, BWORD, CWORD : INT;
		MYSTR: STRING[10] ;
	END_VAR
END_PROGRAM

(* ---- t17-6.st ---- *)
PROGRAM Test
	VAR THREE :
		ARRAY[1..5,1..10,1..8] OF INT;
	END_VAR
END_PROGRAM

(* ---- t17-7.st ---- *)
PROGRAM Test
	VAR RETAIN RTBT:
  		ARRAY[1..2,1..3] OF INT;
	END_VAR
END_PROGRAM

(* ---- t17-8.st ---- *)
PROGRAM Test
	VAR MODULE_8_CONFIG :
   		ANALOG_16_INPUT_CONFIGURATION;
	END_VAR
END_PROGRAM

(* ---- t18-1.st ---- *)
PROGRAM Test
	VAR AT %QX5.1 : BOOL :=1;
          AT %MW6 : INT := 8 ;
	END_VAR
END_PROGRAM

(* ---- t18-10.st ---- *)
PROGRAM Test
	VAR TempLoop :
	  PID :=
	 (PropBand := 2.5,
	  Integral := T#5s);
	END_VAR
END_PROGRAM

(* ---- t18-2.st ---- *)
PROGRAM Test
	VAR RETAIN
  		AT %QW5 : WORD  := 16#FF00 ;
	END_VAR
END_PROGRAM

(* ---- t18-3.st ---- *)
PROGRAM Test
	VAR
   		VALVE_POS AT %QW28 :  INT := 100;
	END_VAR
END_PROGRAM

(* ---- t18-4.st ---- *)
PROGRAM Test
	VAR OUTARY AT %QW6 :
 		ARRAY[0..9] OF INT := [10(1)];
	END_VAR
END_PROGRAM

(* ---- t18-5.st ---- *)
PROGRAM Test
	VAR
  		MYBIT : BOOL := 1 ;
  		OKAY : STRING[10] := 'OK';
	END_VAR
END_PROGRAM

(* ---- t18-6.st ---- *)
PROGRAM Test
	VAR
		BITS : ARRAY[0..7]
			OF BOOL := [1,1,0,0,0,1,0,0] ;
	  	TBT : ARRAY [1..2,1..3]
	        OF INT := [1,2,3(4),6] ;
	END_VAR
END_PROGRAM

(* ---- t18-7.st ---- *)
PROGRAM Test
	VAR RETAIN RTBT :
  		ARRAY(1..2,1..3) OF INT
      		:= [1,2,3(4)];
	END_VAR
END_PROGRAM

(* ---- t18-8.st ---- *)
PROGRAM Test
	VAR MODULE_8_CONFIG:
	  ANALOG_16_INPUT_CONFIGURATION :=
	    (SIGNAL_TYPE := DIFFERENTIAL,
	      CHANNEL
	        := [4((RANGE := UNIPOLAR_1_5V)),
	            (RANGE:= BIPOLAR_10_V,
	             MIN_SCALE := 0,
	             MAX_SCALE := 500)]);
	END_VAR
END_PROGRAM

(* ---- t18-9.st ---- *)
PROGRAM Test
	VAR CONSTANT PI : REAL := 3.141592 ; END_VAR
END_PROGRAM
